INTERFACE I_NodePrototypeVisitor

METHOD VisitNodePrototype
VAR_INPUT
	VisitingPrototype : I_NodePrototype;
END_VAR
END_METHOD

END_INTERFACE

(* stored: Version 1.1.0.1, ProductVersion 3.1.4024.12
   Itf I_NodePrototypeVisitor: Id {2b679aaf-7c54-4be4-9584-ffd5d2a99092}
   Method VisitNodePrototype: Id {76214092-af3e-4a27-911e-657f672a2ded} *)
